{attribute 'qualified_only'}
VAR_GLOBAL PERSISTENT
	
	(* System Settings *) //---------------------------------------------------------------------------------------------- 
	sysRevNumber				: INT;
	sLastSysSettingsChangedBy 	: STRING(256);
	sLastSysSettingsChangedOn 	: STRING(256);
	
	stMachineParam				: ST_HMIParameters;						// Motion Parameters to be used on the software
	stCalibParameters 			: ST_CalibrationSettings;				// Calibration Parameters to be used on the software
	stPumpParameters			: ST_PumpSettings;						// Pump Parameters to be used on the software
	stLeakTestParameters		: ST_LeakTestSettings;					// Leak Test Parameters to be used on the software
	stSolventsInfo	 			: ARRAY[1..4] OF ST_SolventsSettings;	// Solvents name and density to be used on the software
	
	bGeneralSealAndPump			: BOOL := FALSE;						// General Settings only parameter SealAndPump
	bDisplayManualControl		: BOOL := FALSE;						// Security Setting parameter Display Manual Control
	bCheckLogonEachRun			: BOOL := FALSE;						// Security Setting parameter Check Logon Each Run
	
	bMeteringSolvent1Done 		: BOOL := FALSE;
	
	(* Scale/Balance comunication *) //-----------------------------------------------------------------------------------
	aBalanceIP		: T_IPv4Addr 	:= '192.168.1.100';	// Scale TCP IP Adress
	nBalancePort	: UINT 			:= 8001;			// TCP port used to communicate with the scale
	
	(* Air Supply Parameters *) //----------------------------------------------------------------------------------------
	rAirSupplyThreshold		: REAL	:= 4.0;
	rAirSupplyTestingTime	: TIME 	:= T#5S;
	
	

END_VAR

(* stored: Version 1.1.0.1, ProductVersion 3.1.4024.15
   GVL GVL_Settings: Id {7fcbda61-1efa-47f4-8a74-d81c27375a8d} *)
